// TIA Portal project "s7_client" (V15)

(* hardware
DEVICE "S7-1200 station_1"  S7-1200 Station
   slot 0: "Rack_0"  S7-1200 Rack  Rack  V1.0
   slot 1: "PLC_1"  CPU 1214C DC/DC/DC  6ES7 214-1AG40-0XB0  V4.2
*)

// ===== PLC "PLC_1"  CPU 1214C DC/DC/DC =====

VAR_GLOBAL   // PLC tag table "Default tag table"
   "System_Byte" AT %MB1 : Byte;
   "FirstScan" AT %M1.0 : Bool;
   "DiagStatusUpdate" AT %M1.1 : Bool;
   "AlwaysTRUE" AT %M1.2 : Bool;
   "AlwaysFALSE" AT %M1.3 : Bool;
   "Clock_Byte" AT %MB0 : Byte;
   "Clock_10Hz" AT %M0.0 : Bool;
   "Clock_5Hz" AT %M0.1 : Bool;
   "Clock_2.5Hz" AT %M0.2 : Bool;
   "Clock_2Hz" AT %M0.3 : Bool;
   "Clock_1.25Hz" AT %M0.4 : Bool;
   "Clock_1Hz" AT %M0.5 : Bool;
   "Clock_0.625Hz" AT %M0.6 : Bool;
   "Clock_0.5Hz" AT %M0.7 : Bool;
   "Tag_1" AT %M3.0 : Bool;
   "Tag_2" AT %Q0.4 : Bool;
   "Tag_3" AT %Q0.7 : Bool;
   "Q0.5" AT %Q0.5 : Bool;
   "Q0.6" AT %Q0.6 : Bool;
   "Q1.0" AT %Q1.0 : Bool;
   "Q1.1" AT %Q1.1 : Bool;
   "Tag_4" AT %M12.0 : Bool;
   "Tag_5" AT %M12.2 : Bool;
   "Tag_6" AT %M12.1 : Bool;
END_VAR

VAR_GLOBAL   // PLC tag table "vatcp_client"
   "connect_tcp_client" AT %M10.0 : Bool;
END_VAR

DATA_BLOCK "web_com"   // DB1
{ S7_Optimized_Access := 'TRUE' }
VERSION : 0.1
   VAR
      tag_bool : Bool;
      tag_int : Int;
      tag_byte : Byte;
      tag_real : Real;
      tag_string : String;
      tag_int_2 : Int;
   END_VAR
BEGIN
END_DATA_BLOCK

DATA_BLOCK "Modbus_tcp_Client"   // DB3
{ S7_Optimized_Access := 'TRUE' }
VERSION : 0.1
   VAR
      Receive_req : Bool;
      receive_disconnect : Bool;
      receive_MB_mode : USInt;
      RECEIVE_CONNECT : TCON_IP_v4;
      TCP_CIENT_DONE : Bool;
      TCP_CLIENT_BUSY : Bool;
      TCP_CLIENT_ERROR : Bool;
      TCP_STATUS : Word;
      TCP_CIENT_DONE_1 : Bool;
      TCP_CLIENT_BUSY_1 : Bool;
      TCP_CLIENT_ERROR_1 : Bool;
      TCP_STATUS_1 : Word;
   END_VAR
BEGIN
   RECEIVE_CONNECT.RemoteAddress.ADDR[1] := 192;
   RECEIVE_CONNECT.RemoteAddress.ADDR[2] := 168;
   RECEIVE_CONNECT.RemoteAddress.ADDR[3] := 0;
   RECEIVE_CONNECT.RemoteAddress.ADDR[4] := 123;
   RECEIVE_CONNECT.RemotePort := 502;
   RECEIVE_CONNECT.InterfaceId := 64;
   RECEIVE_CONNECT.ID := 1;
   RECEIVE_CONNECT.ActiveEstablished := TRUE;
   RECEIVE_CONNECT.ConnectionType := 11;
END_DATA_BLOCK

DATA_BLOCK "DATA_TCP"   // DB4
{ S7_Optimized_Access := 'FALSE' }
VERSION : 0.1
   VAR
      VALUE : Array[0..9] of Int;
      WRITE : Array[0..9] of Int;
   END_VAR
BEGIN
END_DATA_BLOCK

// folder: System blocks/Program resources

DATA_BLOCK "IEC_Timer_0_DB"   // DB5
{ S7_Optimized_Access := 'TRUE' }
AUTHOR : Simatic
FAMILY : IEC
NAME : IEC_TMR
VERSION : 1.0
// stored: InstanceOfName IEC_TIMER
"IEC_TIMER"
BEGIN
END_DATA_BLOCK

DATA_BLOCK "IEC_Timer_0_DB_1"   // DB6
{ S7_Optimized_Access := 'TRUE' }
AUTHOR : Simatic
FAMILY : IEC
NAME : IEC_TMR
VERSION : 1.0
// stored: InstanceOfName IEC_TIMER
"IEC_TIMER"
BEGIN
END_DATA_BLOCK

DATA_BLOCK "IEC_Timer_0_DB_2"   // DB7
{ S7_Optimized_Access := 'TRUE' }
AUTHOR : Simatic
FAMILY : IEC
NAME : IEC_TMR
VERSION : 1.0
// stored: InstanceOfName IEC_TIMER
"IEC_TIMER"
BEGIN
END_DATA_BLOCK

DATA_BLOCK "IEC_Timer_0_DB_3"   // DB8
{ S7_Optimized_Access := 'TRUE' }
AUTHOR : Simatic
FAMILY : IEC
NAME : IEC_TMR
VERSION : 1.0
// stored: InstanceOfName IEC_TIMER
"IEC_TIMER"
BEGIN
END_DATA_BLOCK

DATA_BLOCK "IEC_Timer_0_DB9"   // DB9
{ S7_Optimized_Access := 'TRUE' }
AUTHOR : Simatic
FAMILY : IEC
NAME : IEC_TMR
VERSION : 1.0
// stored: InstanceOfName IEC_TIMER
"IEC_TIMER"
BEGIN
END_DATA_BLOCK

DATA_BLOCK "IEC_Timer_0_DB_10"   // DB10
{ S7_Optimized_Access := 'TRUE' }
AUTHOR : Simatic
FAMILY : IEC
NAME : IEC_TMR
VERSION : 1.0
// stored: InstanceOfName IEC_TIMER
"IEC_TIMER"
BEGIN
END_DATA_BLOCK

// folder: (top level)

ORGANIZATION_BLOCK "Main"   // OB1, LAD, ProgramCycle
TITLE = "Main Program Sweep (Cycle)"
{ S7_Optimized_Access := 'TRUE' }
VERSION : 0.1
   VAR_INPUT
      Initial_Call : Bool;   // Initial call of this OB
      Remanence : Bool;   // =True, if remanent data are available
   END_VAR
   VAR_TEMP   // added for the SCL form of the ladder/FBD networks
      _w1 : Bool;
      _w2 : Bool;
      _w3 : Bool;
   END_VAR
BEGIN

REGION Network 1
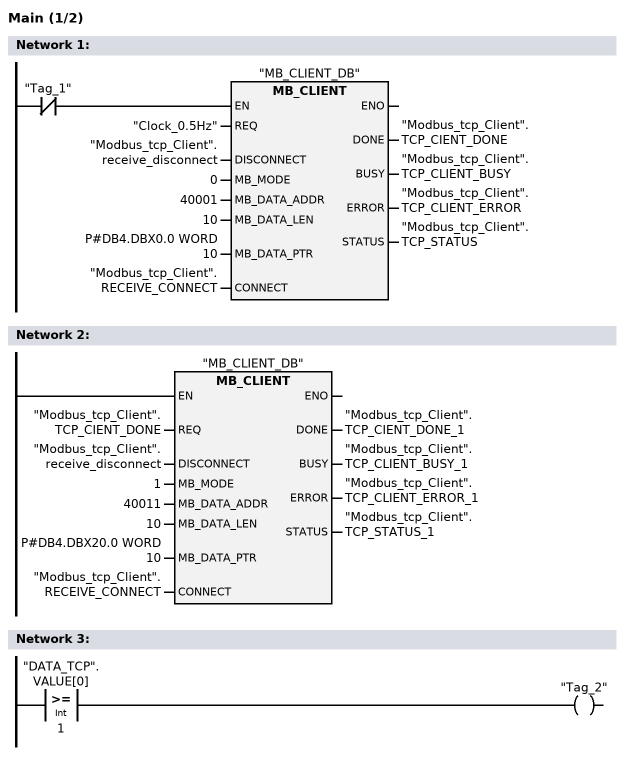
   IF NOT "Tag_1" THEN
       "MB_CLIENT_DB"(REQ := "Clock_0.5Hz",   // MB_CLIENT
                      DISCONNECT := "Modbus_tcp_Client".receive_disconnect,
                      MB_MODE := 0,
                      MB_DATA_ADDR := 40001,
                      MB_DATA_LEN := 10,
                      MB_DATA_PTR := P#DB4.DBX0.0 WORD 10,
                      CONNECT := "Modbus_tcp_Client".RECEIVE_CONNECT,
                      DONE => "Modbus_tcp_Client".TCP_CIENT_DONE,
                      BUSY => "Modbus_tcp_Client".TCP_CLIENT_BUSY,
                      ERROR => "Modbus_tcp_Client".TCP_CLIENT_ERROR,
                      STATUS => "Modbus_tcp_Client".TCP_STATUS);
   END_IF;
END_REGION

REGION Network 2
   "MB_CLIENT_DB"(REQ := "Modbus_tcp_Client".TCP_CIENT_DONE,   // MB_CLIENT
                  DISCONNECT := "Modbus_tcp_Client".receive_disconnect,
                  MB_MODE := 1,
                  MB_DATA_ADDR := 40011,
                  MB_DATA_LEN := 10,
                  MB_DATA_PTR := P#DB4.DBX20.0 WORD 10,
                  CONNECT := "Modbus_tcp_Client".RECEIVE_CONNECT,
                  DONE => "Modbus_tcp_Client".TCP_CIENT_DONE_1,
                  BUSY => "Modbus_tcp_Client".TCP_CLIENT_BUSY_1,
                  ERROR => "Modbus_tcp_Client".TCP_CLIENT_ERROR_1,
                  STATUS => "Modbus_tcp_Client".TCP_STATUS_1);
END_REGION

REGION Network 3
   RUNG wire#powerrail
      { S7_Templates := "SrcType := Int" } GE_Contact(in1 := "DATA_TCP".VALUE[0], in2 := 1)
      Coil( "Tag_2" )
   END_RUNG
   // the same network as SCL:
   "Tag_2" := "DATA_TCP".VALUE[0] >= 1;
END_REGION

REGION Network 4
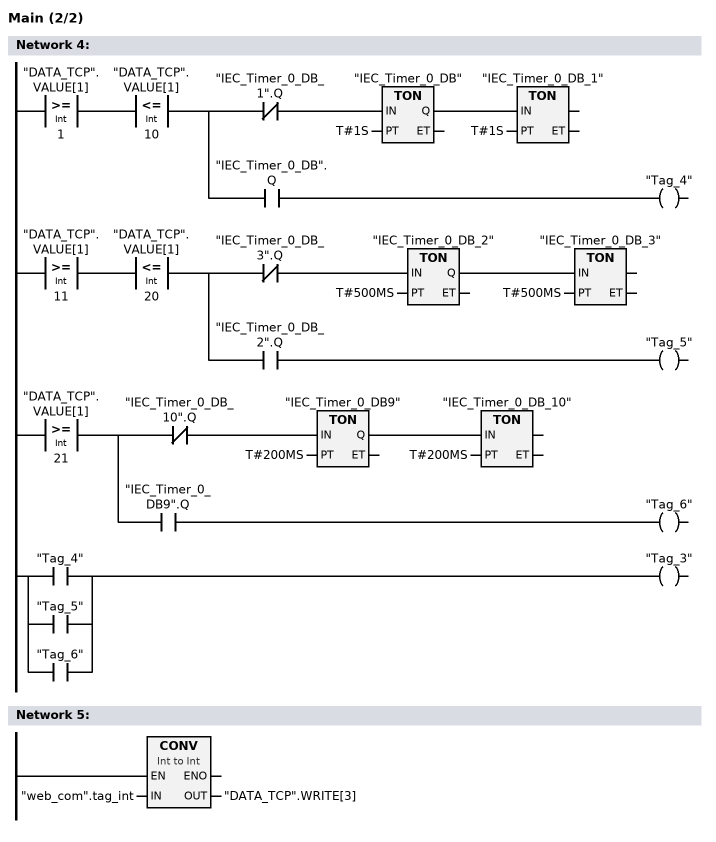
   #_w1 := ("DATA_TCP".VALUE[1] >= 1) AND ("DATA_TCP".VALUE[1] <= 10);
   "IEC_Timer_0_DB".TON(IN := #_w1 AND NOT "IEC_Timer_0_DB_1".Q, PT := T#1S);
   "IEC_Timer_0_DB_1".TON(IN := "IEC_Timer_0_DB".Q, PT := T#1S);
   "Tag_4" := #_w1 AND "IEC_Timer_0_DB".Q;
   #_w2 := ("DATA_TCP".VALUE[1] >= 11) AND ("DATA_TCP".VALUE[1] <= 20);
   "IEC_Timer_0_DB_2".TON(IN := #_w2 AND NOT "IEC_Timer_0_DB_3".Q, PT := T#500MS);
   "IEC_Timer_0_DB_3".TON(IN := "IEC_Timer_0_DB_2".Q, PT := T#500MS);
   "Tag_5" := #_w2 AND "IEC_Timer_0_DB_2".Q;
   #_w3 := "DATA_TCP".VALUE[1] >= 21;
   "IEC_Timer_0_DB9".TON(IN := #_w3 AND NOT "IEC_Timer_0_DB_10".Q, PT := T#200MS);
   "IEC_Timer_0_DB_10".TON(IN := "IEC_Timer_0_DB9".Q, PT := T#200MS);
   "Tag_6" := #_w3 AND "IEC_Timer_0_DB9".Q;
   "Tag_3" := "Tag_4" OR "Tag_5" OR "Tag_6";
END_REGION

REGION Network 5
   RUNG wire#powerrail
      { S7_Templates := "[SrcType := Int, DestType := Int]" } Convert(in := "web_com".tag_int, out => "DATA_TCP".WRITE[3])
   END_RUNG
   // the same network as SCL:
   "DATA_TCP".WRITE[3] := INT_TO_INT("web_com".tag_int);
END_REGION
END_ORGANIZATION_BLOCK